INTERFACE I_SessionIdGenerator

METHOD PUBLIC Generate : T_MAXSTRING
VAR_INPUT
END_VAR
END_METHOD

END_INTERFACE

(* stored: Version 1.1.0.1, ProductVersion 3.1.4024.12
   Itf I_SessionIdGenerator: Id {671b0e78-6011-4b83-b865-f42893b999ed}
   Method Generate: Id {c7ff3c80-3e74-4f2f-9e69-9f17b398f273} *)
